// TIA Portal V19 export
TYPE "type_teachPara_ngConveyor"
// stored: Access Published
   STRUCT
      U2Em4Cm2 { S7_SetPoint := 'True'} : "type_teachPara_axis";   // Yaxis
      U1Em4Cm2 { S7_SetPoint := 'True'} : "type_teachPara_axis";   // Yaxis
   END_STRUCT;
   // // U2Em4Cm2.position[0] : 电芯 放下位置
   // // U1Em4Cm2.position[0] : 电芯 放下位置
END_TYPE
